(* PLC project twetrttr, hty luckyyou 1 *)
(* stored: creationDateTime 2025-03-10T15:45:21, modificationDateTime 2025-03-20T16:54:43 *)

FUNCTION_BLOCK FB0
  VAR
    out1 : INT;
    TON0 : TON;
  END_VAR
  VAR_EXTERNAL
    con1 : BOOL;
  END_VAR

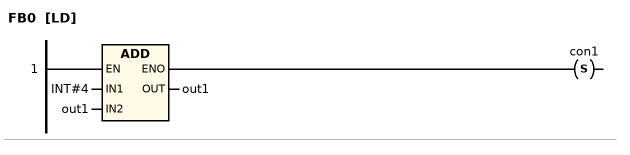
(* LD diagram, written out as Structured Text *)
out1 := INT#4 + out1;
IF TRUE THEN con1 := TRUE; END_IF;
END_FUNCTION_BLOCK

FUNCTION_BLOCK func
  VAR_INPUT
    in1 : BOOL;
  END_VAR
  VAR
    TON0 : TON;
  END_VAR
  VAR_EXTERNAL
    norm1 : BOOL;
  END_VAR

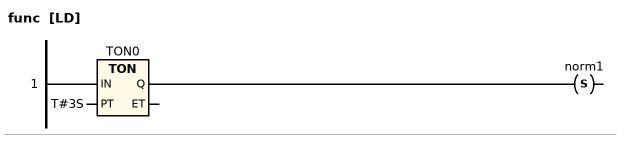
(* LD diagram, written out as Structured Text *)
TON0(IN := TRUE, PT := T#3S);
IF TON0.Q THEN norm1 := TRUE; END_IF;
END_FUNCTION_BLOCK

PROGRAM PLC_PRG
  VAR
    cur : INT;
    out1 : INT;
    FB00 : FB0;
    var1 : INT;
    bool1 : BOOL;
    func_FC : func;
  END_VAR
  VAR_EXTERNAL
    con1 : BOOL;
  END_VAR

            FB00();

IF con1 THEN
FB00();
END_IF;
var1:=1;
var1:=var1*3;
func_FC (in1:=bool1);

          
END_PROGRAM

CONFIGURATION Config0
  RESOURCE Res0 ON PLC
    VAR_GLOBAL RETAIN
      con1 AT %MB131072 : BOOL := TRUE;
    END_VAR
    VAR_GLOBAL CONSTANT
      con2 : BOOL;
    END_VAR
    VAR_GLOBAL
      norm1 : BOOL;
    END_VAR
    TASK task0(INTERVAL := T#20ms, PRIORITY := 0);
    PROGRAM instance0 WITH task0 : PLC_PRG;
  END_RESOURCE
END_CONFIGURATION
